FUNCTION F_MonthString : STRING
VAR_INPUT
	x : WORD;
END_VAR
VAR
	z : INT;
	y : STRING(3);
END_VAR

// --- Simple Month converter: From 1,2,3 to Jan, Fev, Mar"

z := WORD_TO_INT(x);

CASE z OF
	
	1:
		y := 'Jan';
	2:
		y := 'Feb';
	3:
		y := 'Mar';
	4:
		y := 'Apr';
	5:
		y := 'May';
	6:
		y := 'Jun';
	7:
		y := 'Jul';
	8:
		y := 'Aug';
	9:
		y := 'Sep';
	10:
		y := 'Oct';
	11:
		y := 'Nov';
	12:
		y := 'Dec';
	ELSE
		y := 'ukn';
END_CASE

F_MonthString := y;

END_FUNCTION

(* stored: Version 1.1.0.1, ProductVersion 3.1.4024.12
   POU F_MonthString: Id {c9da9571-50c8-4563-8b7a-e76bd7014d92}, SpecialFunc None *)
